FUNCTION_BLOCK FB_ADS_CleanProcess EXTENDS FB_AdsBlockBase
VAR
  // ---------------------------------
  // ADS interface block specific
  sO_Message                 : ST_ADS_MSG_IF;    (*Messaging*)

  (*User commands - Trigger operation*)
  bI_StartCapping            : BOOL := FALSE;
  bO_StartCappingCanEx       : BOOL := FALSE;
  bO_StartCappingExec        : BOOL := FALSE;
                             
  bI_StopCapping             : BOOL := FALSE;
  bO_StopCappingCanEx        : BOOL := FALSE;
  bO_StopCappingExec         : BOOL := FALSE;
                             
  bI_Purge                   : BOOL := FALSE;
  bO_PurgeCanEx              : BOOL := FALSE;
  bO_PurgeExec               : BOOL := FALSE;
                             
  bI_Clean                   : BOOL := FALSE;
  bO_CleanCanEx              : BOOL := FALSE;
  bO_CleanExec               : BOOL := FALSE;
                             
  bI_Maintenance             : BOOL := FALSE;
  bO_MaintenanceCanEx        : BOOL := FALSE;
  bO_MaintenanceExec         : BOOL := FALSE;
                             
  bI_OpenShutter             : BOOL := FALSE;
  bO_OpenShutterCanEx        : BOOL := FALSE;
  bO_OpenShutterExec         : BOOL := FALSE;
                             
  bI_Abort                   : BOOL := FALSE;
  bO_AbortCanEx              : BOOL := FALSE;
  bO_AbortExec               : BOOL := FALSE;

  bI_AcknowledgeError        : BOOL := FALSE;
  bO_AcknowledgeErrorCanEx   : BOOL := FALSE;
  bO_AcknowledgeErrorExec    : BOOL := FALSE;

  (*User settings - State operation*)
  bI_AutoMode                : BOOL := TRUE;  (*del*)
  bI_CleanAfterCapp          : BOOL := FALSE;
  bI_CleanAfterPurge         : BOOL := FALSE;
  bI_PurgeAfterCapp          : BOOL := FALSE; (*del*)
  bI_MaintenanceMode         : BOOL := FALSE;
                             
  (*Flags*)                  
  bO_Busy                    : BOOL;
  bO_Ready                   : BOOL;
  bO_ServiceEnabled          : BOOL;
  bO_AxisProcessMovingVisible: BOOL := TRUE;  (*Cleaning process axis moving is shown at PUC*)
                             
  (*Message Queue - TODO update*)
  bI_FaultAck                : BOOL := FALSE;
  wO_ErrorCode               : WORD;
END_VAR

VAR PERSISTENT
  nR_Pattern                 : UDINT;  (*check pattern for rem validity*)
END_VAR

PROPERTY bAcknowledgeError : BOOL
SET
bI_AcknowledgeError := bAcknowledgeError;
END_SET
END_PROPERTY

METHOD config
VAR_INPUT
  aName                     : STRING;
  bAxisProcessMovingVisible : BOOL;  
END_VAR
aO_Name                     := aName;

bO_AxisProcessMovingVisible := bAxisProcessMovingVisible;
END_METHOD

METHOD PROTECTED initRemVar
VAR_INPUT
END_VAR
(*load default initial values if pattern was invalid*)
IF nR_Pattern <> 16#ABCD THEN
  ;
ELSE  
  nR_Pattern      := 16#ABCD;
END_IF

(*Init values*)
END_METHOD

METHOD ResetCommands : BOOL
VAR_INPUT
END_VAR
bI_StartCapping := FALSE;
bI_StopCapping  := FALSE;
bI_Maintenance  := FALSE;
bI_Clean        := FALSE;
bI_Purge        := FALSE;
END_METHOD

METHOD setFeedback
VAR_INPUT
  bStartCappingCanEx       : BOOL; 
  bStartCappingExec        : BOOL;  

  bStopCappingCanEx        : BOOL;  
  bStopCappingExec         : BOOL;  

  bPurgeCanEx              : BOOL; 
  bPurgeExec               : BOOL;  

  bCleanCanEx              : BOOL; 
  bCleanExec               : BOOL;  

  bMaintenanceCanEx        : BOOL;  
  bMaintenanceExec         : BOOL;  

  bOpenShutterCanEx        : BOOL;  
  bOpenShutterExec         : BOOL;  

  bAbortCanEx              : BOOL; 
  bAbortExec               : BOOL;  

  bAcknowledgeErrorCanEx   : BOOL;  
  bAcknowledgeErrorExec    : BOOL;  

  bBusy                    : BOOL; 
  bReady                   : BOOL; 
  bServiceEnabled          : BOOL; 
  bAxisProcessMovingVisible: BOOL; 

  wErrorCode               : WORD; 
END_VAR
bO_StartCappingCanEx       := bStartCappingCanEx;
bO_StartCappingExec        := bStartCappingExec;

bO_StopCappingCanEx        := bStopCappingCanEx;
bO_StopCappingExec         := bStopCappingExec;

bO_PurgeCanEx              := bPurgeCanEx;
bO_PurgeExec               := bPurgeExec;

bO_CleanCanEx              := bCleanCanEx;
bO_CleanExec               := bCleanExec;

bO_MaintenanceCanEx        := bMaintenanceCanEx;
bO_MaintenanceExec         := bMaintenanceExec;

bO_OpenShutterCanEx        := bOpenShutterCanEx;
bO_OpenShutterExec         := bOpenShutterExec;

bO_AbortCanEx              := bAbortCanEx;
bO_AbortExec               := bAbortExec;

bO_AcknowledgeErrorCanEx   := bAcknowledgeErrorCanEx;
bO_AcknowledgeErrorExec    := bAcknowledgeErrorExec;

bO_Busy                    := bBusy;
bO_Ready                   := bReady;
bO_ServiceEnabled          := bServiceEnabled;
bO_AxisProcessMovingVisible:= bAxisProcessMovingVisible;

wO_ErrorCode               := wErrorCode;
END_METHOD

(*
  Setup constant ADS Block definitions.
  HOWTO: in abstract implmentation call
      init(aVersion:=, aType:=, nType:=, eLayer:=);
*)
METHOD  setup
init( aVersion := '01.00.01'
    , aType    := 'CleanProcess'
    , nType    := eMa_BLK_MACHINE
    , eLayer   := E_AdsLayer.Structural);
END_METHOD

PROPERTY sMsgInterface : POINTER TO ST_ADS_MSG_IF
GET
sMsgInterface := ADR(sO_Message);
END_GET
END_PROPERTY

END_FUNCTION_BLOCK

(* stored: Version 1.1.0.1, ProductVersion 3.1.4024.11
   POU FB_ADS_CleanProcess: Id {02fdcc45-2cbf-46ed-b4e2-51b235b39c44}, SpecialFunc None
   Property bAcknowledgeError: Id {c8a7df29-9919-4093-857e-372271473b5c}
   Set Set: Id {bb358ce5-b877-433a-8189-23e41fdc691a}
   Method config: Id {cfff9820-f309-44a9-b29f-f4982e59276f}
   Method initRemVar: Id {e2282e57-c61f-4d5e-be3d-ba65f82a666a}
   Method ResetCommands: Id {b16dda10-aded-4d78-a0a9-f4273d287851}
   Method setFeedback: Id {8d8f3ff0-5d37-4971-8db5-60faacc470bd}
   Method setup: Id {b9929b56-48a6-4347-b167-83c786449c9c}
   Property sMsgInterface: Id {de7432b2-f6d5-4a61-83ad-17a5b2f39c40}
   Get Get: Id {71c74738-03e2-4406-9a78-18e6ba115832} *)
